// SIMATIC S7-200 project (STEP 7-Micro/WIN), CPU 226 REL 02.01

SYMBOL_TABLE 用户定义1
仓泵投入             I0.0
仓泵退出             I0.1
灰库高料位1           I2.7
灰库高料位2           I3.0
灰库高料位3           I3.1
进1库允许            I2.4
进2库允许            I2.5
进3库允许            I2.6
仓泵出料阀2           Q0.7
仓泵就地自动1          I1.6
气源压力上限           I1.5
仓泵压力下限           I0.6
仓泵就地料位1          I2.2
仓泵进料时间1          I1.2
仓泵出料阀1           Q0.6
仓泵输送阀1           Q0.4
仓泵排气阀1           Q0.2
仓泵进料阀1           Q0.0
仓泵就地复位1          I2.0
报警复位             I0.5
料满1              Q1.4
仓泵投入标志位          M2.4
仓泵运行标志位          M2.3
仓泵就地复位           M2.0
一号库开标志位          M8.3
二号库开标志位          M8.4
三号库开标志位          M8.5
一号库料位高报          M8.0
二号库料位高报          M8.1
三号库料位高报          M8.2
汽源压力下限           M0.7
输送阀运行超时1         M1.1
输送阀运行超时2         M1.2
堵管               M2.1
END_SYMBOL_TABLE

ORGANIZATION_BLOCK 程序块:OB1
TITLE=程序注释
BEGIN
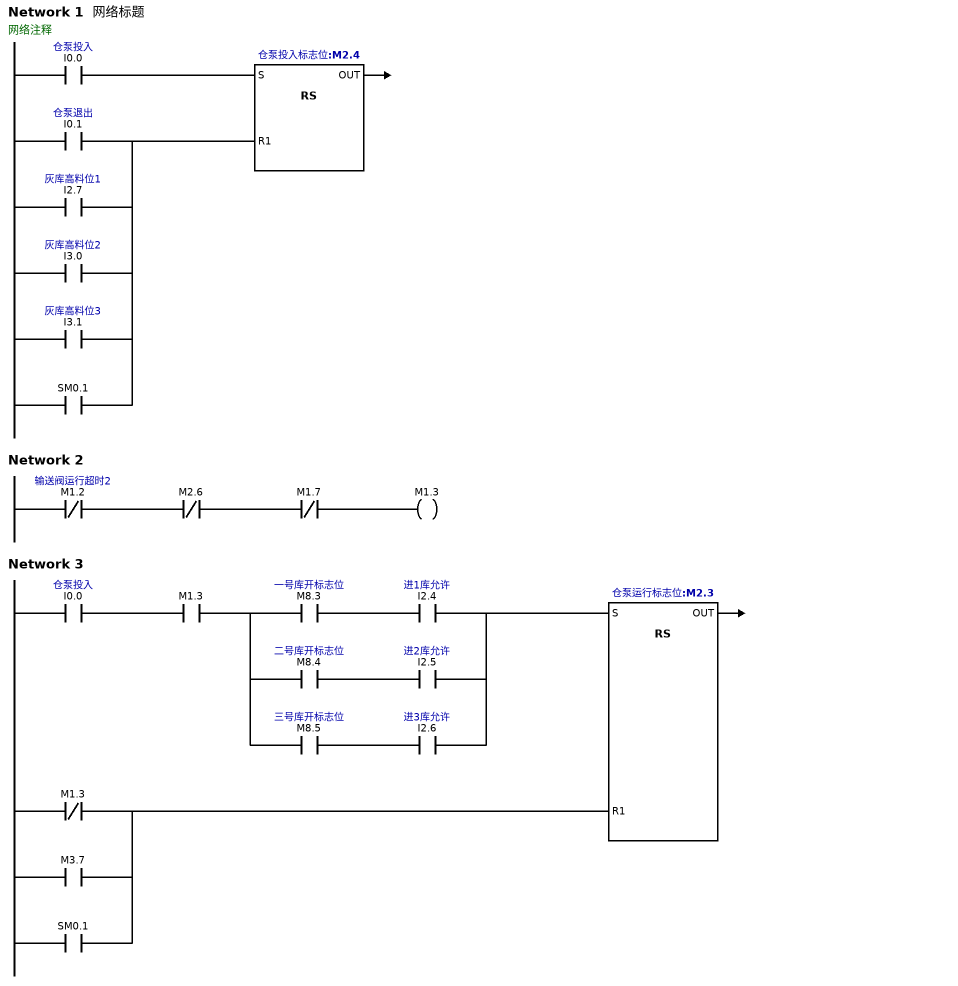
Network 1 // 网络标题
// 网络注释
// (network saved uncompiled; LAD cells follow)
// row 0: c0 -| |- 仓泵投入:I0.0  c1 --  c2 [RS 仓泵投入标志位:M2.4 S:=power@row0, R1:=power@row1, OUT=>power]  c3 ->
// row 1: c0 -| |- 仓泵退出:I0.1 v  c1 --  c2 [box]
// row 2: c0 -| |- 灰库高料位1:I2.7 ^v
// row 3: c0 -| |- 灰库高料位2:I3.0 ^v
// row 4: c0 -| |- 灰库高料位3:I3.1 ^v
// row 5: c0 -| |- SM0.1 ^
Network 2
LDN    输送阀运行超时2:M1.2
AN     M2.6
AN     M1.7
=      M1.3
Network 3
LD     仓泵投入:I0.0
A      M1.3
LD     一号库开标志位:M8.3
A      进1库允许:I2.4
LD     二号库开标志位:M8.4
A      进2库允许:I2.5
OLD
LD     三号库开标志位:M8.5
A      进3库允许:I2.6
OLD
ALD
LDN    M1.3
O      M3.7
O      SM0.1
NOT
LPS
A      仓泵运行标志位:M2.3
=      仓泵运行标志位:M2.3
LPP
ALD
O      仓泵运行标志位:M2.3
=      仓泵运行标志位:M2.3
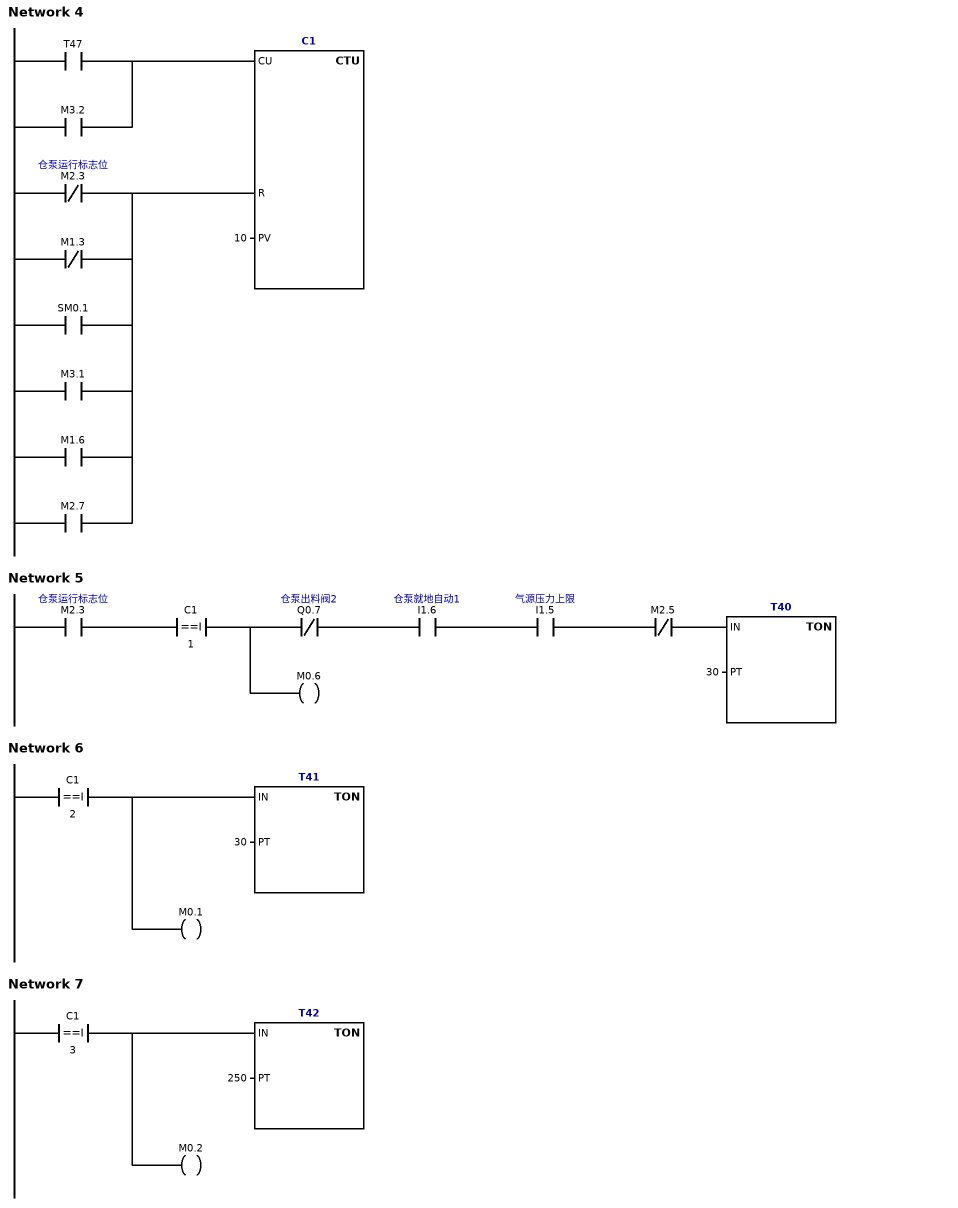
Network 4
LD     T47
O      M3.2
LDN    仓泵运行标志位:M2.3
ON     M1.3
O      SM0.1
O      M3.1
O      M1.6
O      M2.7
CTU    C1, 10
Network 5
// (network saved uncompiled; LAD cells follow)
// row 0: c0 -| |- 仓泵运行标志位:M2.3  c1 -|==I|- C1, 1 v  c2 -|/|- 仓泵出料阀2:Q0.7  c3 -| |- 仓泵就地自动1:I1.6  c4 -| |- 气源压力上限:I1.5  c5 -|/|- M2.5  c6 [TON T40 IN:=power@row0, PT:=30]
// row 1: c1 ^  c2 -( ) M0.6  c6 [box]
Network 6
// (network saved uncompiled; LAD cells follow)
// row 0: c0 -|==I|- C1, 2 v  c1 --  c2 [TON T41 IN:=power@row0, PT:=30]
// row 1: c0 ^v  c2 [box]
// row 2: c0 ^  c1 -( ) M0.1
Network 7
// (network saved uncompiled; LAD cells follow)
// row 0: c0 -|==I|- C1, 3 v  c1 --  c2 [TON T42 IN:=power@row0, PT:=250]
// row 1: c0 ^v  c2 [box]
// row 2: c0 ^  c1 -( ) M0.2
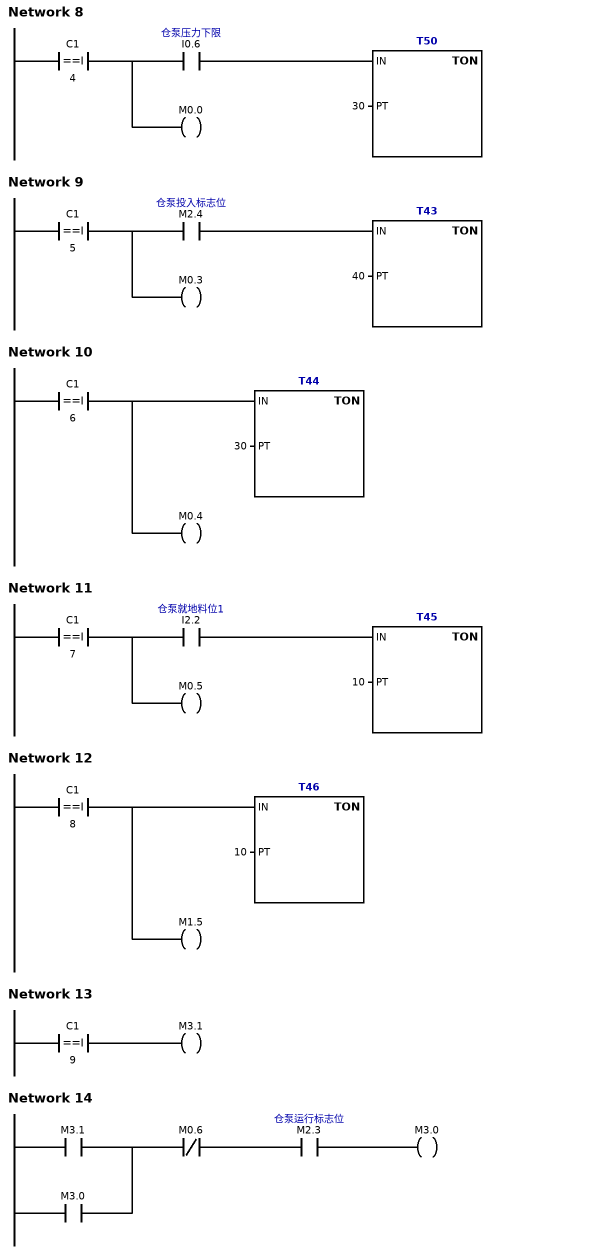
Network 8
// (network saved uncompiled; LAD cells follow)
// row 0: c0 -|==I|- C1, 4 v  c1 -| |- 仓泵压力下限:I0.6  c2 --  c3 [TON T50 IN:=power@row0, PT:=30]
// row 1: c0 ^  c1 -( ) M0.0  c3 [box]
Network 9
// (network saved uncompiled; LAD cells follow)
// row 0: c0 -|==I|- C1, 5 v  c1 -| |- 仓泵投入标志位:M2.4  c2 --  c3 [TON T43 IN:=power@row0, PT:=40]
// row 1: c0 ^  c1 -( ) M0.3  c3 [box]
Network 10
// (network saved uncompiled; LAD cells follow)
// row 0: c0 -|==I|- C1, 6 v  c1 --  c2 [TON T44 IN:=power@row0, PT:=30]
// row 1: c0 ^v  c2 [box]
// row 2: c0 ^  c1 -( ) M0.4
Network 11
// (network saved uncompiled; LAD cells follow)
// row 0: c0 -|==I|- C1, 7 v  c1 -| |- 仓泵就地料位1:I2.2  c2 --  c3 [TON T45 IN:=power@row0, PT:=10]
// row 1: c0 ^  c1 -( ) M0.5  c3 [box]
Network 12
// (network saved uncompiled; LAD cells follow)
// row 0: c0 -|==I|- C1, 8 v  c1 --  c2 [TON T46 IN:=power@row0, PT:=10]
// row 1: c0 ^v  c2 [box]
// row 2: c0 ^  c1 -( ) M1.5
Network 13
// (network saved uncompiled; LAD cells follow)
// row 0: c0 -|==I|- C1, 9  c1 -( ) M3.1
Network 14
// (network saved uncompiled; LAD cells follow)
// row 0: c0 -| |- M3.1 v  c1 -|/|- M0.6  c2 -| |- 仓泵运行标志位:M2.3  c3 -( ) M3.0
// row 1: c0 -| |- M3.0 ^
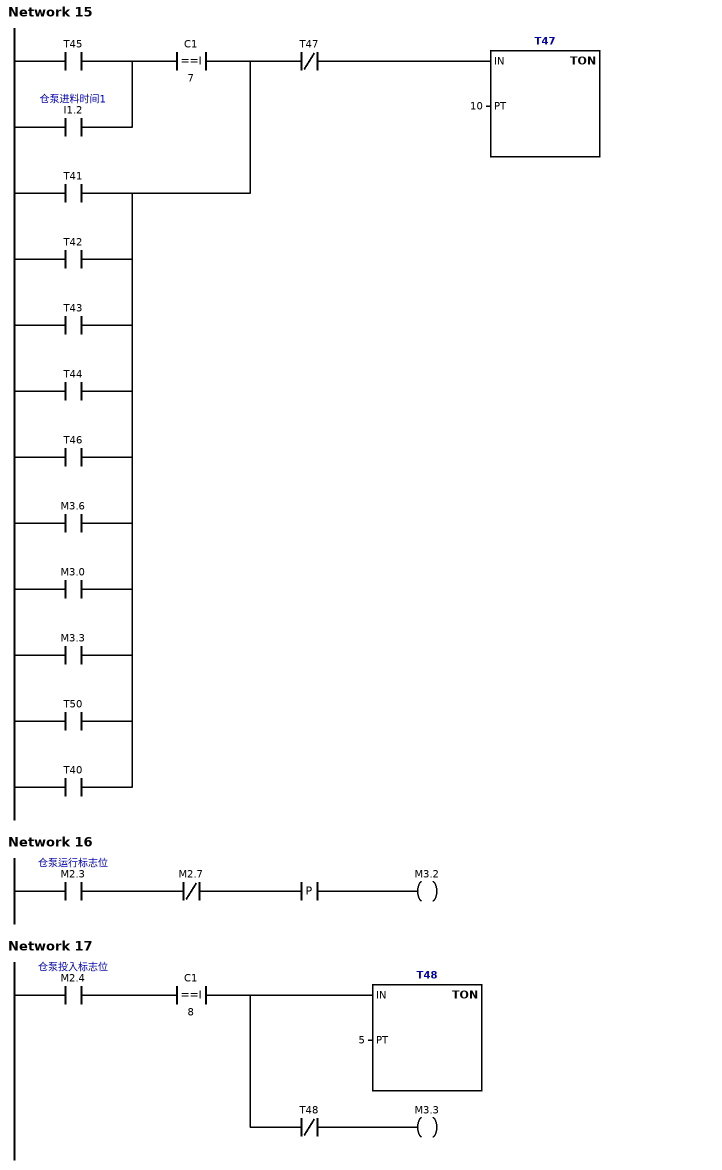
Network 15
// (network saved uncompiled; LAD cells follow)
// row 0: c0 -| |- T45 v  c1 -|==I|- C1, 7 v  c2 -|/|- T47  c3 --  c4 [TON T47 IN:=power@row0, PT:=10]
// row 1: c0 -| |- 仓泵进料时间1:I1.2 ^  c1 ^v  c4 [box]
// row 2: c0 -| |- T41 v  c1 -- ^
// row 3: c0 -| |- T42 ^v
// row 4: c0 -| |- T43 ^v
// row 5: c0 -| |- T44 ^v
// row 6: c0 -| |- T46 ^v
// row 7: c0 -| |- M3.6 ^v
// row 8: c0 -| |- M3.0 ^v
// row 9: c0 -| |- M3.3 ^v
// row 10: c0 -| |- T50 ^v
// row 11: c0 -| |- T40 ^
Network 16
// (network saved uncompiled; LAD cells follow)
// row 0: c0 -| |- 仓泵运行标志位:M2.3  c1 -|/|- M2.7  c2 -|P|-  c3 -( ) M3.2
Network 17
// (network saved uncompiled; LAD cells follow)
// row 0: c0 -| |- 仓泵投入标志位:M2.4  c1 -|==I|- C1, 8 v  c2 --  c3 [TON T48 IN:=power@row0, PT:=5]
// row 1: c1 ^v  c3 [box]
// row 2: c1 ^  c2 -|/|- T48  c3 -( ) M3.3
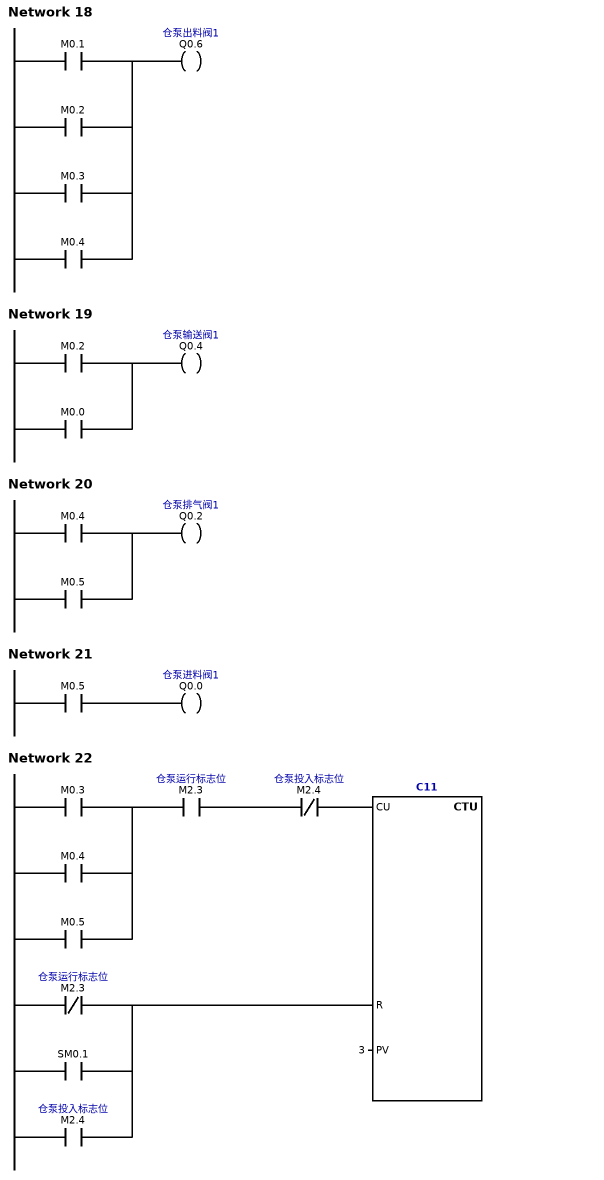
Network 18
// (network saved uncompiled; LAD cells follow)
// row 0: c0 -| |- M0.1 v  c1 -( ) 仓泵出料阀1:Q0.6
// row 1: c0 -| |- M0.2 ^v
// row 2: c0 -| |- M0.3 ^v
// row 3: c0 -| |- M0.4 ^
Network 19
// (network saved uncompiled; LAD cells follow)
// row 0: c0 -| |- M0.2 v  c1 -( ) 仓泵输送阀1:Q0.4
// row 1: c0 -| |- M0.0 ^
Network 20
// (network saved uncompiled; LAD cells follow)
// row 0: c0 -| |- M0.4 v  c1 -( ) 仓泵排气阀1:Q0.2
// row 1: c0 -| |- M0.5 ^
Network 21
// (network saved uncompiled; LAD cells follow)
// row 0: c0 -| |- M0.5  c1 -( ) 仓泵进料阀1:Q0.0
Network 22
// (network saved uncompiled; LAD cells follow)
// row 0: c0 -| |- M0.3 v  c1 -| |- 仓泵运行标志位:M2.3  c2 -|/|- 仓泵投入标志位:M2.4  c3 [CTU C11 CU:=power@row0, R:=power@row3, PV:=3]
// row 1: c0 -| |- M0.4 ^v  c3 [box]
// row 2: c0 -| |- M0.5 ^  c3 [box]
// row 3: c0 -|/|- 仓泵运行标志位:M2.3 v  c1 --  c2 --  c3 [box]
// row 4: c0 -| |- SM0.1 ^v  c3 [box]
// row 5: c0 -| |- 仓泵投入标志位:M2.4 ^
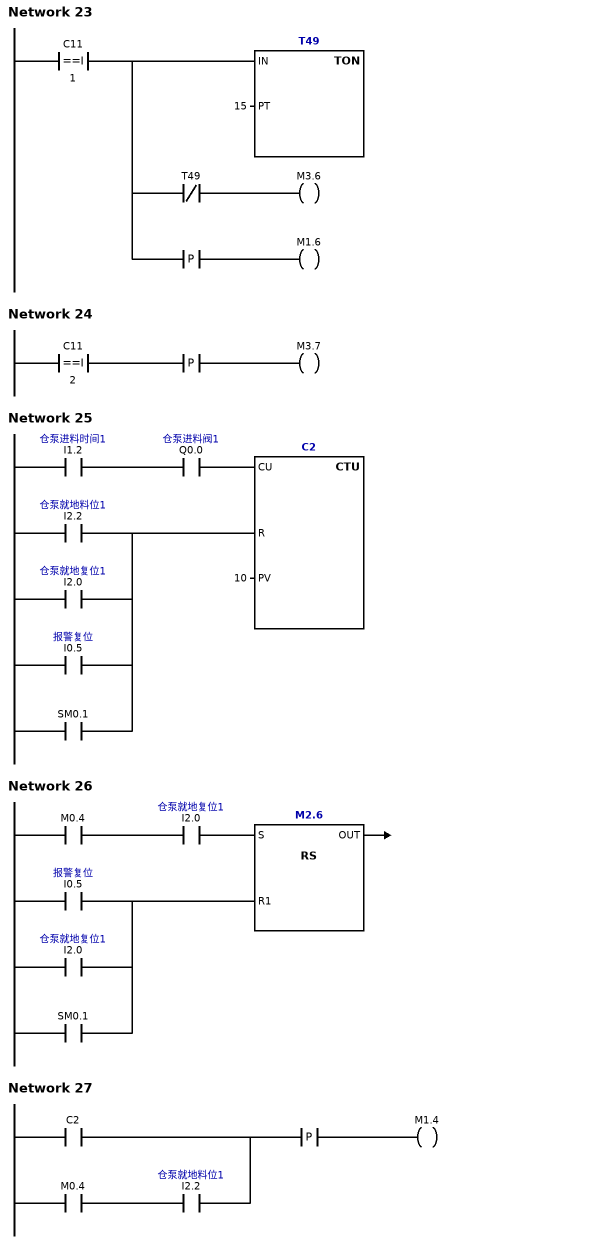
Network 23
// (network saved uncompiled; LAD cells follow)
// row 0: c0 -|==I|- C11, 1 v  c1 --  c2 [TON T49 IN:=power@row0, PT:=15]
// row 1: c0 ^v  c2 [box]
// row 2: c0 ^v  c1 -|/|- T49  c2 -( ) M3.6
// row 3: c0 ^  c1 -|P|-  c2 -( ) M1.6
Network 24
// (network saved uncompiled; LAD cells follow)
// row 0: c0 -|==I|- C11, 2  c1 -|P|-  c2 -( ) M3.7
Network 25
// (network saved uncompiled; LAD cells follow)
// row 0: c0 -| |- 仓泵进料时间1:I1.2  c1 -| |- 仓泵进料阀1:Q0.0  c2 [CTU C2 CU:=power@row0, R:=power@row1, PV:=10]
// row 1: c0 -| |- 仓泵就地料位1:I2.2 v  c1 --  c2 [box]
// row 2: c0 -| |- 仓泵就地复位1:I2.0 ^v  c2 [box]
// row 3: c0 -| |- 报警复位:I0.5 ^v
// row 4: c0 -| |- SM0.1 ^
Network 26
// (network saved uncompiled; LAD cells follow)
// row 0: c0 -| |- M0.4  c1 -| |- 仓泵就地复位1:I2.0  c2 [RS M2.6 S:=power@row0, R1:=power@row1, OUT=>power]  c3 ->
// row 1: c0 -| |- 报警复位:I0.5 v  c1 --  c2 [box]
// row 2: c0 -| |- 仓泵就地复位1:I2.0 ^v
// row 3: c0 -| |- SM0.1 ^
Network 27
// (network saved uncompiled; LAD cells follow)
// row 0: c0 -| |- C2  c1 -- v  c2 -|P|-  c3 -( ) M1.4
// row 1: c0 -| |- M0.4  c1 -| |- 仓泵就地料位1:I2.2 ^
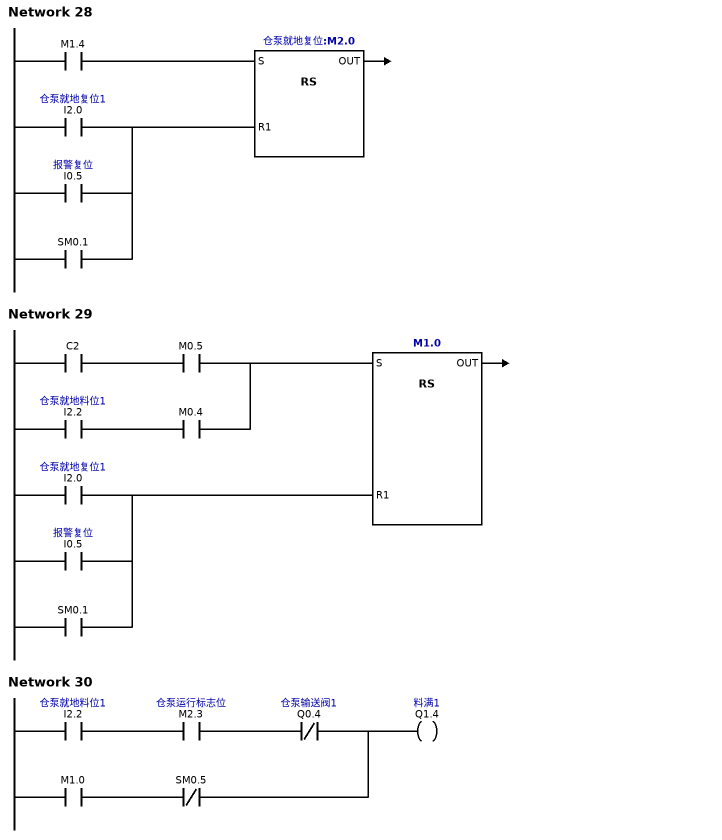
Network 28
// (network saved uncompiled; LAD cells follow)
// row 0: c0 -| |- M1.4  c1 --  c2 [RS 仓泵就地复位:M2.0 S:=power@row0, R1:=power@row1, OUT=>power]  c3 ->
// row 1: c0 -| |- 仓泵就地复位1:I2.0 v  c1 --  c2 [box]
// row 2: c0 -| |- 报警复位:I0.5 ^v
// row 3: c0 -| |- SM0.1 ^
Network 29
// (network saved uncompiled; LAD cells follow)
// row 0: c0 -| |- C2  c1 -| |- M0.5 v  c2 --  c3 [RS M1.0 S:=power@row0, R1:=power@row2, OUT=>power]  c4 ->
// row 1: c0 -| |- 仓泵就地料位1:I2.2  c1 -| |- M0.4 ^  c3 [box]
// row 2: c0 -| |- 仓泵就地复位1:I2.0 v  c1 --  c2 --  c3 [box]
// row 3: c0 -| |- 报警复位:I0.5 ^v
// row 4: c0 -| |- SM0.1 ^
Network 30
// (network saved uncompiled; LAD cells follow)
// row 0: c0 -| |- 仓泵就地料位1:I2.2  c1 -| |- 仓泵运行标志位:M2.3  c2 -|/|- 仓泵输送阀1:Q0.4 v  c3 -( ) 料满1:Q1.4
// row 1: c0 -| |- M1.0  c1 -|/|- SM0.5  c2 -- ^
END_ORGANIZATION_BLOCK
